// TIA Portal V17 export
// export: Created 2024-08-09T12:53:14.4278295Z, ExportSetting WithDefaults, DisplayName Totally Integrated Automation Portal, DisplayVersion V17 Update 7, DisplayName TIA Portal Openness, DisplayVersion V17 Update 7, DisplayName TIA Portal Version Control Interface, DisplayVersion V17, DisplayName STEP 7 Professional, DisplayVersion V17 Update 7, DisplayName STEP 7 Safety, DisplayVersion V17 Update 6, DisplayName WinCC Professional, DisplayVersion V17 Update 7
VAR_GLOBAL   // PLC tag table "Verse_Sac"
END_VAR
VAR_GLOBAL CONSTANT   // user constants
   NIV_VS_DEBUT_LOT : USInt := 1;
   NIV_VS_VIDANGE_PES_PARTIELLE : USInt := 10;
   NIV_VS_FIN_INCOR : USInt := 30;
   NIV_VS_DEBUT_VIDANGE : USInt := 50;
   NIV_VS_FIN_SYNCHRO : USInt := 70;
   NIV_VS_FIN_VIDANGE : USInt := 90;
   NIV_VS_FIN_LOT : USInt := 255;
END_VAR
